{attribute addProperty BoxType "EL6201-0000-0017"}
{attribute addProperty Id "Slave_27A_DI0BIT10.125209Slave_27A_DI1BIT10.125210Slave_27A_DI2BIT10.125211Slave_27A_DI3BIT10.125212Slave_27B_DI0BIT10.125213Slave_27B_DI1BIT10.125214Slave_27B_DI2BIT10.125215Slave_27B_DI3BIT10.125216"}
{attribute addProperty CRC "49157180"}
{attribute addProperty SizeInBites "8"}
{attribute addProperty SizeInBytes "1"}
TYPE Slave_27_Inputs_02EE143C :
STRUCT
	{attribute addProperty Name "Slave_27A_DI0"}
	Slave_27A_DI0 : BIT;
	{attribute addProperty Name "Slave_27A_DI1"}
	Slave_27A_DI1 : BIT;
	{attribute addProperty Name "Slave_27A_DI2"}
	Slave_27A_DI2 : BIT;
	{attribute addProperty Name "Slave_27A_DI3"}
	Slave_27A_DI3 : BIT;
	{attribute addProperty Name "Slave_27B_DI0"}
	Slave_27B_DI0 : BIT;
	{attribute addProperty Name "Slave_27B_DI1"}
	Slave_27B_DI1 : BIT;
	{attribute addProperty Name "Slave_27B_DI2"}
	Slave_27B_DI2 : BIT;
	{attribute addProperty Name "Slave_27B_DI3"}
	Slave_27B_DI3 : BIT;
END_STRUCT
END_TYPE

(* stored: Version 1.2.0.0, ProductVersion 3.1.4024.9
   DUT Slave_27_Inputs_02EE143C: Id {eeca9fbb-79fb-4353-ba02-adec368310b4} *)
